// TIA Portal V21 export
TYPE "Rcp_Cmd_Type"
   STRUCT
      Load_in_Work : Bool;   // Load recipe in work (changeover)
      Load_in_Edit : Bool;   // Load recipe in edit recipe
      Load_in_Edit_from_work : Bool;   // Load recipe in edit from work recipe
      Save_in_Archive : Bool;   // Save recipe in archive
      Save_in_Work : Bool;   // Save recipe in work recipe (update)
      Copy : Bool;   // Copy recipe
      Reload_RCP_GEN_List : Bool;   // Updates the RCP_GEN_list of the recipes generic data reading from the archive
      Reset : Bool;   // Alarm reset from machine
   END_STRUCT;
END_TYPE
